% RSLogix 500 project SOL6.RSS, saved by version 8.30.00.16 %
PROJECT "PROJ6"    % processor: Bul.1763 MicroLogix 1100 Series B %

PROGRAM FILES
  LAD 2   9 rungs

DATA FILES
  O0 OUTPUT  4 elements
  I1 INPUT  6 elements
  S2 STATUS  66 elements
  B3 BINARY  1 elements
  T4 TIMER  1 elements
  C5 COUNTER  4 elements
  R6 CONTROL  1 elements
  N7 INTEGER  4 elements
  F8 FLOAT  1 elements

LADDER 2
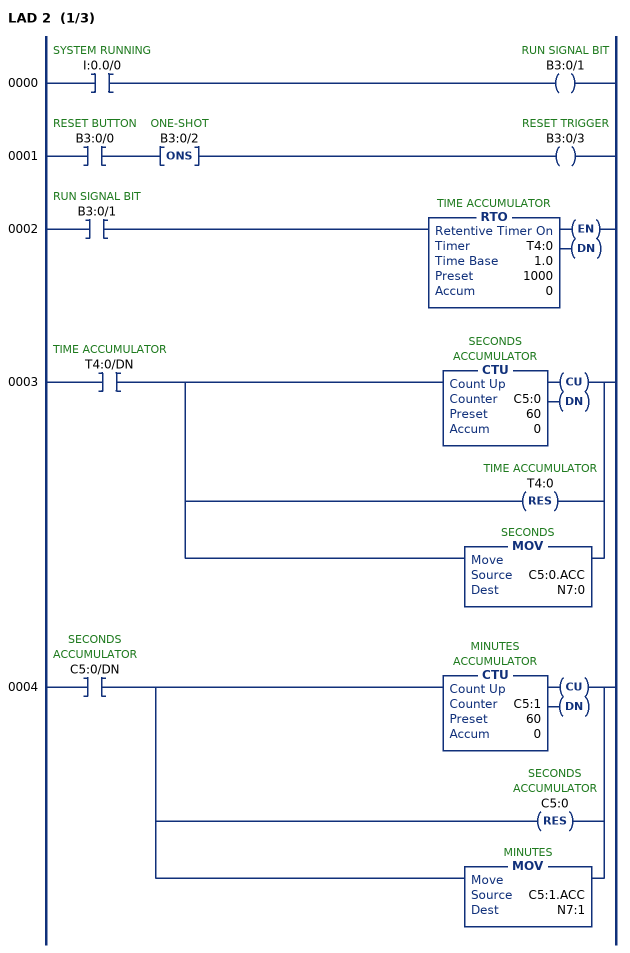
% Rung: 0 %
SOR XIC I:0.0/0 OTE B3:0/1 EOR
%   I:0.0/0  "SYSTEM RUNNING" %
%   B3:0/1  "RUN SIGNAL BIT" %
% Rung: 1 %
SOR XIC B3:0/0 ONS B3:0/2 OTE B3:0/3 EOR
%   B3:0/0  "RESET BUTTON" %
%   B3:0/2  "ONE-SHOT" %
%   B3:0/3  "RESET TRIGGER" %
% Rung: 2 %
SOR XIC B3:0/1 RTO T4:0 1.0 1000 0 EOR
%   B3:0/1  "RUN SIGNAL BIT" %
%   T4:0  "TIME ACCUMULATOR" %
% Rung: 3 %
SOR XIC T4:0/DN BST CTU C5:0 60 0 NXB RES T4:0 NXB MOV C5:0.ACC N7:0 BND EOR
%   T4:0  "TIME ACCUMULATOR" %
%   C5:0  "SECONDS ACCUMULATOR" %
%   N7:0  "SECONDS" %
% Rung: 4 %
SOR XIC C5:0/DN BST CTU C5:1 60 0 NXB RES C5:0 NXB MOV C5:1.ACC N7:1 BND EOR
%   C5:0  "SECONDS ACCUMULATOR" %
%   C5:1  "MINUTES ACCUMULATOR" %
%   N7:1  "MINUTES" %

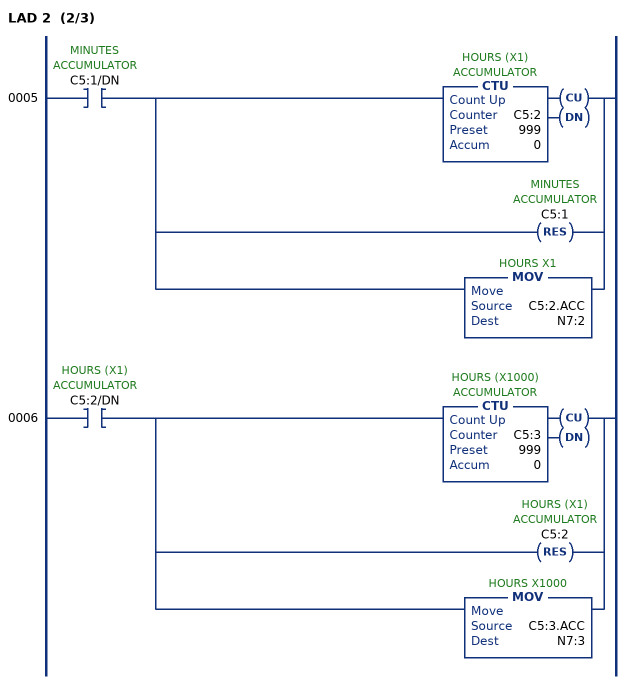
% Rung: 5 %
SOR XIC C5:1/DN BST CTU C5:2 999 0 NXB RES C5:1 NXB MOV C5:2.ACC N7:2 BND EOR
%   C5:1  "MINUTES ACCUMULATOR" %
%   C5:2  "HOURS (X1) ACCUMULATOR" %
%   N7:2  "HOURS X1" %
% Rung: 6 %
SOR XIC C5:2/DN BST CTU C5:3 999 0 NXB RES C5:2 NXB MOV C5:3.ACC N7:3 BND EOR
%   C5:2  "HOURS (X1) ACCUMULATOR" %
%   C5:3  "HOURS (X1000) ACCUMULATOR" %
%   N7:3  "HOURS X1000" %

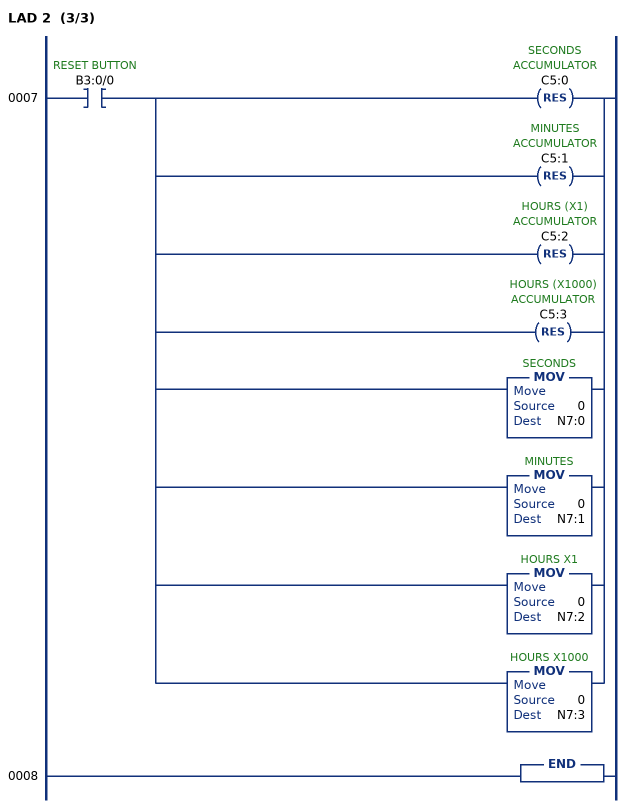
% Rung: 7 %
SOR XIC B3:0/0 BST RES C5:0 NXB RES C5:1 NXB RES C5:2 NXB RES C5:3 NXB MOV 0 N7:0 NXB MOV 0 N7:1 NXB MOV 0 N7:2 NXB MOV 0 N7:3 BND EOR
%   B3:0/0  "RESET BUTTON" %
%   C5:0  "SECONDS ACCUMULATOR" %
%   C5:1  "MINUTES ACCUMULATOR" %
%   C5:2  "HOURS (X1) ACCUMULATOR" %
%   C5:3  "HOURS (X1000) ACCUMULATOR" %
%   N7:0  "SECONDS" %
%   N7:1  "MINUTES" %
%   N7:2  "HOURS X1" %
%   N7:3  "HOURS X1000" %
% Rung: 8 %
SOR END EOR

DATA TABLE (non-zero values as saved)
DATA T4
% .PRE .ACC %
% T4:0 % 1000 0
DATA C5
% .PRE .ACC %
% C5:0 % 60 0
% C5:1 % 60 0
% C5:2 % 999 0
% C5:3 % 999 0
